DATA_BLOCK "dbArchiveAutoConveyor"
{ S7_Optimized_Access := 'TRUE' }
VERSION : 0.8
NON_RETAIN
"fbArchiveAutoConveyor"

BEGIN

END_DATA_BLOCK

